{attribute 'GeneratedUsingTerminal: EK1100-0000-0018'}
{attribute addProperty BoxType "EK1100-0000-0018"}
{attribute addProperty Id "Beckhoff_EQ1xxxEK1122Beckhoff_EQ1xxxEK1122_0186272478"}
{attribute addProperty CRC "4156720697"}
{attribute addProperty Size "78"}
TYPE Beckhoff_EQ1xxx_F7C28639 EXTENDS EK1100_AB5A9467 :
STRUCT
	{attribute addProperty Name "Beckhoff_EQ1xxxEK1122"}
	{attribute addProperty PreviousPort "Beckhoff EQ1xxx : B"}
	Beckhoff_EQ1xxxEK1122 : Beckhoff_EQ1xxxEK1122_01862724;
END_STRUCT
END_TYPE

(* stored: Version 1.2.0.0, ProductVersion 3.1.4024.9
   DUT Beckhoff_EQ1xxx_F7C28639: Id {4b0a5bad-9694-424c-b15a-eefd20580381} *)
